Fanuc KAREL source: kt00100.KL

-- PROVISIONAL review KL for V940-1; original PC SHA256 1fed10cfd48f2f4a27548f1c6644bb40007fcffa65e782c30f03feb002d44069
-- Incomplete behavior may be omitted. Consult companion uncertainty JSON. Do not deploy.
PROGRAM KT00100
%NOLOCKGROUP
VAR
  I1 : INTEGER
  R2 : REAL
  OUT : REAL
BEGIN
  -- V9_ZERO_TABLE_METADATA_HINT layout=0001; no indexed target words; source/name/runtime held
  -- UNRESOLVED_PC offsets 5-16; opcodes 2E,23
  -- UNRESOLVED_PC offsets 21-32; opcodes 2E,23
  -- UNRESOLVED_PC offsets 37-59; opcodes 21,21,29,64,29,6C,23
  -- UNRESOLVED_PC offsets 64-68; opcodes 7F
END KT00100
